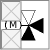
VISUALIZATION Icon_ML_AB_Up  // 50x50
VAR_INPUT
    ITF_STELLANTRIEB_IN   :   ITF_STELLANTRIEB;	
END_VAR
    Frame (4,16 18x18)
        shows Motor(ITF_STELLANTRIEB_IN := ITF_STELLANTRIEB_IN)
    Frame (20,9 24x32)
        shows ML_Ventil_AB_Up(rProzent := ITF_STELLANTRIEB_IN.proOnY)
    Image (1,1 20x20), invisible if: NOT ITF_STELLANTRIEB_IN.proIsWarning, image: CtaVisSymbols.ImagePool.CtaWarning
    Image (1,29 20x20), invisible if: NOT ITF_STELLANTRIEB_IN.proIsHandOnOrOff, image: CtaVisSymbols.ImagePool.front_hand_Yellow
    Image (1,29 20x20), invisible if: NOT ITF_STELLANTRIEB_IN.proHandOff, image: CtaVisSymbols.ImagePool.front_hand_Yellow_Off
END_VISUALIZATION

// 40 Visualizations/ICON/StellAntrieb_BASE/Icons/Motor_Left/Icon_ML_Verteiler
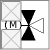
VISUALIZATION Icon_ML_Verteiler  // 50x50
VAR_INPUT
    ITF_STELLANTRIEB_IN   :   ITF_STELLANTRIEB;	
END_VAR
    Frame (4,16 18x18)
        shows Motor(ITF_STELLANTRIEB_IN := ITF_STELLANTRIEB_IN)
    Frame (20,9 24x32)
        shows ML_Ventil_Verteiler(rProzent := ITF_STELLANTRIEB_IN.proOnY)
    Image (1,1 20x20), invisible if: NOT ITF_STELLANTRIEB_IN.proIsWarning, image: CtaVisSymbols.ImagePool.CtaWarning
    Image (1,29 20x20), invisible if: NOT ITF_STELLANTRIEB_IN.proIsHandOnOrOff, image: CtaVisSymbols.ImagePool.front_hand_Yellow
    Image (1,29 20x20), invisible if: NOT ITF_STELLANTRIEB_IN.proHandOff, image: CtaVisSymbols.ImagePool.front_hand_Yellow_Off
END_VISUALIZATION

// 40 Visualizations/ICON/StellAntrieb_BASE/Icons/Motor_Left/Icon_ML_Durchfluss
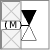
VISUALIZATION Icon_ML_Durchfluss  // 50x50
VAR_INPUT
    ITF_STELLANTRIEB_IN   :   ITF_STELLANTRIEB;	
END_VAR
    Frame (4,16 18x18)
        shows Motor(ITF_STELLANTRIEB_IN := ITF_STELLANTRIEB_IN)
    Frame (20,9 17x32)
        shows ML_Durchgang(rProzent := ITF_STELLANTRIEB_IN.proOnY)
    Image (1,1 20x20), invisible if: NOT ITF_STELLANTRIEB_IN.proIsWarning, image: CtaVisSymbols.ImagePool.CtaWarning
    Image (1,29 20x20), invisible if: NOT ITF_STELLANTRIEB_IN.proIsHandOnOrOff, image: CtaVisSymbols.ImagePool.front_hand_Yellow
    Image (1,29 20x20), invisible if: NOT ITF_STELLANTRIEB_IN.proHandOff, image: CtaVisSymbols.ImagePool.front_hand_Yellow_Off
END_VISUALIZATION

// 40 Visualizations/ICON/StellAntrieb_BASE/Icons/Motor_Right/Icon_MR_AB_Down
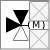
VISUALIZATION Icon_MR_AB_Down  // 50x50
VAR_INPUT
    ITF_STELLANTRIEB_IN   :   ITF_STELLANTRIEB;	
END_VAR
    Frame (27,16 18x18)
        shows Motor(ITF_STELLANTRIEB_IN := ITF_STELLANTRIEB_IN)
    Frame (5,9 24x32)
        shows MR_Ventil_AB_Down(rProzent := ITF_STELLANTRIEB_IN.proOnY)
    Image (29,1 20x20), invisible if: NOT ITF_STELLANTRIEB_IN.proIsWarning, image: CtaVisSymbols.ImagePool.CtaWarning
    Image (29,29 20x20), invisible if: NOT ITF_STELLANTRIEB_IN.proIsHandOnOrOff, image: CtaVisSymbols.ImagePool.front_hand_Yellow
    Image (29,29 20x20), invisible if: NOT ITF_STELLANTRIEB_IN.proHandOff, image: CtaVisSymbols.ImagePool.front_hand_Yellow_Off
END_VISUALIZATION

// 40 Visualizations/ICON/StellAntrieb_BASE/Icons/Motor_Right/Icon_MR_AB_Up
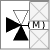
VISUALIZATION Icon_MR_AB_Up  // 50x50
VAR_INPUT
    ITF_STELLANTRIEB_IN   :   ITF_STELLANTRIEB;	
END_VAR
    Frame (27,16 18x18)
        shows Motor(ITF_STELLANTRIEB_IN := ITF_STELLANTRIEB_IN)
    Frame (5,9 24x32)
        shows MR_Ventil_AB_Up(rProzent := ITF_STELLANTRIEB_IN.proOnY)
    Image (29,1 20x20), invisible if: NOT ITF_STELLANTRIEB_IN.proIsWarning, image: CtaVisSymbols.ImagePool.CtaWarning
    Image (29,29 20x20), invisible if: NOT ITF_STELLANTRIEB_IN.proIsHandOnOrOff, image: CtaVisSymbols.ImagePool.front_hand_Yellow
    Image (29,29 20x20), invisible if: NOT ITF_STELLANTRIEB_IN.proHandOff, image: CtaVisSymbols.ImagePool.front_hand_Yellow_Off
END_VISUALIZATION

// 40 Visualizations/ICON/StellAntrieb_BASE/Icons/Motor_Right/Icon_MR_Durchfluss
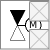
VISUALIZATION Icon_MR_Durchfluss  // 50x50
VAR_INPUT
    ITF_STELLANTRIEB_IN   :   ITF_STELLANTRIEB;	
END_VAR
    Frame (24,16 18x18)
        shows Motor(ITF_STELLANTRIEB_IN := ITF_STELLANTRIEB_IN)
    Frame (9,9 17x32)
        shows MR_Durchgang(rProzent := ITF_STELLANTRIEB_IN.proOnY)
    Image (29,1 20x20), invisible if: NOT ITF_STELLANTRIEB_IN.proIsWarning, image: CtaVisSymbols.ImagePool.CtaWarning
    Image (29,29 20x20), invisible if: NOT ITF_STELLANTRIEB_IN.proIsHandOnOrOff, image: CtaVisSymbols.ImagePool.front_hand_Yellow
    Image (29,29 20x20), invisible if: NOT ITF_STELLANTRIEB_IN.proHandOff, image: CtaVisSymbols.ImagePool.front_hand_Yellow_Off
END_VISUALIZATION

// 40 Visualizations/ICON/StellAntrieb_BASE/Icons/Motor_Right/Icon_MR_Verteiler
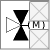
VISUALIZATION Icon_MR_Verteiler  // 50x50
VAR_INPUT
    ITF_STELLANTRIEB_IN   :   ITF_STELLANTRIEB;	
END_VAR
    Frame (27,16 18x18)
        shows Motor(ITF_STELLANTRIEB_IN := ITF_STELLANTRIEB_IN)
    Frame (5,9 24x32)
        shows MR_Ventil_Verteiler(rProzent := ITF_STELLANTRIEB_IN.proOnY)
    Image (29,1 20x20), invisible if: NOT ITF_STELLANTRIEB_IN.proIsWarning, image: CtaVisSymbols.ImagePool.CtaWarning
    Image (29,29 20x20), invisible if: NOT ITF_STELLANTRIEB_IN.proIsHandOnOrOff, image: CtaVisSymbols.ImagePool.front_hand_Yellow
    Image (29,29 20x20), invisible if: NOT ITF_STELLANTRIEB_IN.proHandOff, image: CtaVisSymbols.ImagePool.front_hand_Yellow_Off
END_VISUALIZATION

// 40 Visualizations/ICON/StellAntrieb_BASE/Icons/Motor_Above/Icon_MA_AB_L
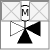
VISUALIZATION Icon_MA_AB_L  // 50x50
VAR_INPUT
    ITF_STELLANTRIEB_IN   :   ITF_STELLANTRIEB;	
END_VAR
    Frame (16,4 18x18)
        shows Motor(ITF_STELLANTRIEB_IN := ITF_STELLANTRIEB_IN)
    Frame (9,20 32x24)
        shows MA_Ventil_AB_L(rProzent := ITF_STELLANTRIEB_IN.proOnY)
    Image (1,1 20x20), invisible if: NOT ITF_STELLANTRIEB_IN.proIsWarning, image: CtaVisSymbols.ImagePool.CtaWarning
    Image (29,1 20x20), invisible if: NOT ITF_STELLANTRIEB_IN.proIsHandOnOrOff, image: CtaVisSymbols.ImagePool.front_hand_Yellow
    Image (29,1 20x20), invisible if: NOT ITF_STELLANTRIEB_IN.proHandOff, image: CtaVisSymbols.ImagePool.front_hand_Yellow_Off
END_VISUALIZATION

// 40 Visualizations/ICON/StellAntrieb_BASE/Icons/Motor_Above/Icon_MA_AB_R
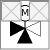
VISUALIZATION Icon_MA_AB_R  // 50x50
VAR_INPUT
    ITF_STELLANTRIEB_IN   :   ITF_STELLANTRIEB;	
END_VAR
    Frame (16,4 18x18)
        shows Motor(ITF_STELLANTRIEB_IN := ITF_STELLANTRIEB_IN)
    Frame (9,20 32x24)
        shows MA_Ventil_AB_R(rProzent := ITF_STELLANTRIEB_IN.proOnY)
    Image (1,1 20x20), invisible if: NOT ITF_STELLANTRIEB_IN.proIsWarning, image: CtaVisSymbols.ImagePool.CtaWarning
    Image (29,1 20x20), invisible if: NOT ITF_STELLANTRIEB_IN.proIsHandOnOrOff, image: CtaVisSymbols.ImagePool.front_hand_Yellow
    Image (29,1 20x20), invisible if: NOT ITF_STELLANTRIEB_IN.proHandOff, image: CtaVisSymbols.ImagePool.front_hand_Yellow_Off
END_VISUALIZATION

// 40 Visualizations/ICON/StellAntrieb_BASE/Icons/Motor_Above/Icon_MA_Durchfluss
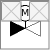
VISUALIZATION Icon_MA_Durchfluss  // 50x50
VAR_INPUT
    ITF_STELLANTRIEB_IN   :   ITF_STELLANTRIEB;	
END_VAR
    Frame (16,4 18x18)
        shows Motor(ITF_STELLANTRIEB_IN := ITF_STELLANTRIEB_IN)
    Frame (9,20 32x17)
        shows MA_Durchgang(rProzent := ITF_STELLANTRIEB_IN.proOnY)
    Image (1,1 20x20), invisible if: NOT ITF_STELLANTRIEB_IN.proIsWarning, image: CtaVisSymbols.ImagePool.CtaWarning
    Image (29,1 20x20), invisible if: NOT ITF_STELLANTRIEB_IN.proIsHandOnOrOff, image: CtaVisSymbols.ImagePool.front_hand_Yellow
    Image (29,1 20x20), invisible if: NOT ITF_STELLANTRIEB_IN.proHandOff, image: CtaVisSymbols.ImagePool.front_hand_Yellow_Off
END_VISUALIZATION

// 40 Visualizations/ICON/StellAntrieb_BASE/Icons/Motor_Above/Icon_MA_Verteiler
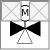
VISUALIZATION Icon_MA_Verteiler  // 50x50
VAR_INPUT
    ITF_STELLANTRIEB_IN   :   ITF_STELLANTRIEB;	
END_VAR
    Frame (16,4 18x18)
        shows Motor(ITF_STELLANTRIEB_IN := ITF_STELLANTRIEB_IN)
    Frame (9,20 32x24)
        shows MA_Ventil_Verteiler(rProzent := ITF_STELLANTRIEB_IN.proOnY)
    Image (1,1 20x20), invisible if: NOT ITF_STELLANTRIEB_IN.proIsWarning, image: CtaVisSymbols.ImagePool.CtaWarning
    Image (29,1 20x20), invisible if: NOT ITF_STELLANTRIEB_IN.proIsHandOnOrOff, image: CtaVisSymbols.ImagePool.front_hand_Yellow
    Image (29,1 20x20), invisible if: NOT ITF_STELLANTRIEB_IN.proHandOff, image: CtaVisSymbols.ImagePool.front_hand_Yellow_Off
END_VISUALIZATION

// 40 Visualizations/ICON/StellAntrieb_BASE/Icons/Motor_Below/Icon_MB_AB_L
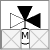
VISUALIZATION Icon_MB_AB_L  // 50x50
VAR_INPUT
    ITF_STELLANTRIEB_IN   :   ITF_STELLANTRIEB;	
END_VAR
    Frame (16,27 18x18)
        shows Motor(ITF_STELLANTRIEB_IN := ITF_STELLANTRIEB_IN)
    Frame (9,5 32x24)
        shows MB_Ventil_AB_L(rProzent := ITF_STELLANTRIEB_IN.proOnY)
    Image (1,29 20x20), invisible if: NOT ITF_STELLANTRIEB_IN.proIsWarning, image: CtaVisSymbols.ImagePool.CtaWarning
    Image (29,29 20x20), invisible if: NOT ITF_STELLANTRIEB_IN.proIsHandOnOrOff, image: CtaVisSymbols.ImagePool.front_hand_Yellow
    Image (29,29 20x20), invisible if: NOT ITF_STELLANTRIEB_IN.proHandOff, image: CtaVisSymbols.ImagePool.front_hand_Yellow_Off
END_VISUALIZATION

// 40 Visualizations/ICON/StellAntrieb_BASE/Icons/Motor_Below/Icon_MB_AB_R
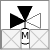
VISUALIZATION Icon_MB_AB_R  // 50x50
VAR_INPUT
    ITF_STELLANTRIEB_IN   :   ITF_STELLANTRIEB;	
END_VAR
    Frame (16,27 18x18)
        shows Motor(ITF_STELLANTRIEB_IN := ITF_STELLANTRIEB_IN)
    Frame (9,5 32x24)
        shows MB_Ventil_AB_R(rProzent := ITF_STELLANTRIEB_IN.proOnY)
    Image (1,29 20x20), invisible if: NOT ITF_STELLANTRIEB_IN.proIsWarning, image: CtaVisSymbols.ImagePool.CtaWarning
    Image (29,29 20x20), invisible if: NOT ITF_STELLANTRIEB_IN.proIsHandOnOrOff, image: CtaVisSymbols.ImagePool.front_hand_Yellow
    Image (29,29 20x20), invisible if: NOT ITF_STELLANTRIEB_IN.proHandOff, image: CtaVisSymbols.ImagePool.front_hand_Yellow_Off
END_VISUALIZATION

// 40 Visualizations/ICON/StellAntrieb_BASE/Icons/Motor_Below/Icon_MB_Verteiler
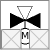
VISUALIZATION Icon_MB_Verteiler  // 50x50
VAR_INPUT
    ITF_STELLANTRIEB_IN   :   ITF_STELLANTRIEB;	
END_VAR
    Frame (16,27 18x18)
        shows Motor(ITF_STELLANTRIEB_IN := ITF_STELLANTRIEB_IN)
    Frame (9,5 32x24)
        shows MB_Ventil_Verteiler(rProzent := ITF_STELLANTRIEB_IN.proOnY)
    Image (1,29 20x20), invisible if: NOT ITF_STELLANTRIEB_IN.proIsWarning, image: CtaVisSymbols.ImagePool.CtaWarning
    Image (29,29 20x20), invisible if: NOT ITF_STELLANTRIEB_IN.proIsHandOnOrOff, image: CtaVisSymbols.ImagePool.front_hand_Yellow
    Image (29,29 20x20), invisible if: NOT ITF_STELLANTRIEB_IN.proHandOff, image: CtaVisSymbols.ImagePool.front_hand_Yellow_Off
END_VISUALIZATION

// 40 Visualizations/ICON/StellAntrieb_BASE/Icons/Motor_Below/Icon_MB_Durchfluss
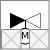
VISUALIZATION Icon_MB_Durchfluss  // 50x50
VAR_INPUT
    ITF_STELLANTRIEB_IN   :   ITF_STELLANTRIEB;	
END_VAR
    Frame (16,27 18x18)
        shows Motor(ITF_STELLANTRIEB_IN := ITF_STELLANTRIEB_IN)
    Frame (9,12 32x17)
        shows MB_Durchgang(rProzent := ITF_STELLANTRIEB_IN.proOnY)
    Image (1,29 20x20), invisible if: NOT ITF_STELLANTRIEB_IN.proIsWarning, image: CtaVisSymbols.ImagePool.CtaWarning
    Image (29,29 20x20), invisible if: NOT ITF_STELLANTRIEB_IN.proIsHandOnOrOff, image: CtaVisSymbols.ImagePool.front_hand_Yellow
    Image (29,29 20x20), invisible if: NOT ITF_STELLANTRIEB_IN.proHandOff, image: CtaVisSymbols.ImagePool.front_hand_Yellow_Off
END_VISUALIZATION

// 40 Visualizations/ICON/StellAntrieb_RIGHT/Motor_Right/Valve_AB_Down/Below/StellAntrieb_MR_Valve_AB_Down_Txt_R_Below
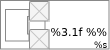
VISUALIZATION StellAntrieb_MR_Valve_AB_Down_Txt_R_Below  // 110x50
VAR_INPUT
    ITF_STELLANTRIEB_IN   	:   ITF_STELLANTRIEB;	
END_VAR
VAR_INPUT CONSTANT
	stExklParameter			:	STRING[40] := '';
END_VAR
VAR CONSTANT
	uiIconNr				: 	UINT := 25;
END_VAR
    Frame (0,0 110x50), invisible if: NOT fcCheckQuerryReturnIcon(_ITF_In := ITF_STELLANTRIEB_IN,_uiIconNr_In := uiIconNr)
        shows StellAntrieb_MR_Valve_AB_Down_RB_CheckQuerry(ITF_STELLANTRIEB_IN := ITF_STELLANTRIEB_IN, stExklParameter := stExklParameter)
        shows Icon()
END_VISUALIZATION

// 40 Visualizations/ICON/StellAntrieb_RIGHT/Motor_Right/Valve_AB_Down/Below/StellAntrieb_MR_Valve_AB_Down_RB_CheckEnabled
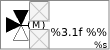
VISUALIZATION StellAntrieb_MR_Valve_AB_Down_RB_CheckEnabled  // 110x50
VAR_INPUT
    ITF_STELLANTRIEB_IN   	:   ITF_STELLANTRIEB;
	stExklParameter			:	STRING[40];
END_VAR
    Frame (0,0 50x50), invisible if: NOT ITF_STELLANTRIEB_IN.proIsEnabled
        shows Icon_MR_AB_Down(ITF_STELLANTRIEB_IN := ITF_STELLANTRIEB_IN)
    Frame (50,25 60x25), invisible if: NOT ITF_STELLANTRIEB_IN.proIsEnabled
        shows ValueDwnUp(ITF_STELLANTRIEB_IN := ITF_STELLANTRIEB_IN, uiTextAusrichtung := 4)
    Rectangle (0,0 110x50)
        OnMouseClick:  Dialog=StellAntrieb_POPUP, Parameters={stExklParameter: stExklParameter, ITF_STELLANTRIEBIN: ITF_STELLANTRIEB_IN, uiPopUpGruppe: 0}, OpenCentered=True
END_VISUALIZATION

// 40 Visualizations/ICON/StellAntrieb_RIGHT/Motor_Right/Valve_AB_Down/Below/StellAntrieb_MR_Valve_AB_Down_RB_CheckQuerry
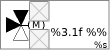
VISUALIZATION StellAntrieb_MR_Valve_AB_Down_RB_CheckQuerry  // 110x50
VAR_INPUT
    ITF_STELLANTRIEB_IN   	:   ITF_STELLANTRIEB;	
	stExklParameter			:	STRING[40];
END_VAR
    Frame (0,0 110x50)
        shows StellAntrieb_MR_Valve_AB_Down_RB_CheckEnabled(ITF_STELLANTRIEB_IN := ITF_STELLANTRIEB_IN, stExklParameter := stExklParameter)
END_VISUALIZATION

// 40 Visualizations/ICON/StellAntrieb_LEFT/Motor_LEFT/Valve_AB_Down/Above/StellAntrieb_ML_Valve_AB_Down_LA_CheckEnabled
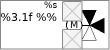
VISUALIZATION StellAntrieb_ML_Valve_AB_Down_LA_CheckEnabled  // 110x50
VAR_INPUT
    ITF_STELLANTRIEB_IN   	:   ITF_STELLANTRIEB;	
	stExklParameter			:	STRING[40];
END_VAR
    Frame (61,0 50x50), invisible if: NOT ITF_STELLANTRIEB_IN.proIsEnabled
        shows Icon_ML_AB_Down(ITF_STELLANTRIEB_IN := ITF_STELLANTRIEB_IN)
    Frame (0,0 60x25), invisible if: NOT ITF_STELLANTRIEB_IN.proIsEnabled
        shows ValueUpDwn(ITF_STELLANTRIEB_IN := ITF_STELLANTRIEB_IN, uiTextAusrichtung := 6)
    Rectangle (0,0 110x50)
        OnMouseClick:  Dialog=StellAntrieb_POPUP, Parameters={stExklParameter: stExklParameter, ITF_STELLANTRIEBIN: ITF_STELLANTRIEB_IN, uiPopUpGruppe: 0}, OpenCentered=True
END_VISUALIZATION

// 40 Visualizations/ICON/StellAntrieb_LEFT/Motor_LEFT/Valve_AB_Down/Above/StellAntrieb_ML_Valve_AB_Down_LA_CheckQuerry
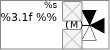
VISUALIZATION StellAntrieb_ML_Valve_AB_Down_LA_CheckQuerry  // 110x50
VAR_INPUT
    ITF_STELLANTRIEB_IN   	:   ITF_STELLANTRIEB;
	stExklParameter			:	STRING[40];
END_VAR
    Frame (0,0 110x50)
        shows StellAntrieb_ML_Valve_AB_Down_LA_CheckEnabled(ITF_STELLANTRIEB_IN := ITF_STELLANTRIEB_IN, stExklParameter := stExklParameter)
END_VISUALIZATION

// 40 Visualizations/ICON/StellAntrieb_LEFT/Motor_LEFT/Valve_AB_Down/Above/StellAntrieb_ML_Valve_AB_Down_Txt_L_Above
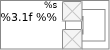
VISUALIZATION StellAntrieb_ML_Valve_AB_Down_Txt_L_Above  // 110x50
VAR_INPUT
    ITF_STELLANTRIEB_IN   	:   ITF_STELLANTRIEB;	
END_VAR
VAR_INPUT CONSTANT
	stExklParameter			:	STRING[40] := '';
END_VAR
VAR CONSTANT
	uiIconNr				: 	UINT := 8;
END_VAR
    Frame (0,0 110x50), invisible if: NOT fcCheckQuerryReturnIcon(_ITF_In := ITF_STELLANTRIEB_IN,_uiIconNr_In := uiIconNr)
        shows StellAntrieb_ML_Valve_AB_Down_LA_CheckQuerry(ITF_STELLANTRIEB_IN := ITF_STELLANTRIEB_IN, stExklParameter := stExklParameter)
        shows Icon()
END_VISUALIZATION

// 40 Visualizations/ICON/StellAntrieb_LEFT/Motor_LEFT/Valve_AB_Down/Below/StellAntrieb_ML_Valve_AB_Down_LB_CheckEnabled
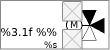
VISUALIZATION StellAntrieb_ML_Valve_AB_Down_LB_CheckEnabled  // 110x50
VAR_INPUT
    ITF_STELLANTRIEB_IN   	:   ITF_STELLANTRIEB;
	stExklParameter			:	STRING[40];
END_VAR
    Frame (61,0 50x50), invisible if: NOT ITF_STELLANTRIEB_IN.proIsEnabled
        shows Icon_ML_AB_Down(ITF_STELLANTRIEB_IN := ITF_STELLANTRIEB_IN)
    Frame (0,25 60x25), invisible if: NOT ITF_STELLANTRIEB_IN.proIsEnabled
        shows ValueDwnUp(ITF_STELLANTRIEB_IN := ITF_STELLANTRIEB_IN, uiTextAusrichtung := 6)
    Rectangle (0,0 110x50)
        OnMouseClick:  Dialog=StellAntrieb_POPUP, Parameters={stExklParameter: stExklParameter, ITF_STELLANTRIEBIN: ITF_STELLANTRIEB_IN, uiPopUpGruppe: 0}, OpenCentered=True
END_VISUALIZATION

// 40 Visualizations/ICON/StellAntrieb_LEFT/Motor_LEFT/Valve_AB_Down/Below/StellAntrieb_ML_Valve_AB_Down_LB_CheckQuerry
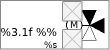
VISUALIZATION StellAntrieb_ML_Valve_AB_Down_LB_CheckQuerry  // 110x50
VAR_INPUT
    ITF_STELLANTRIEB_IN   	:   ITF_STELLANTRIEB;
	stExklParameter			:	STRING[40];
END_VAR
    Frame (0,0 110x50)
        shows StellAntrieb_ML_Valve_AB_Down_LB_CheckEnabled(ITF_STELLANTRIEB_IN := ITF_STELLANTRIEB_IN, stExklParameter := stExklParameter)
END_VISUALIZATION

// 40 Visualizations/ICON/StellAntrieb_LEFT/Motor_LEFT/Valve_AB_Down/Below/StellAntrieb_ML_Valve_AB_Down_Txt_L_Below
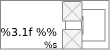
VISUALIZATION StellAntrieb_ML_Valve_AB_Down_Txt_L_Below  // 110x50
VAR_INPUT
    ITF_STELLANTRIEB_IN   	:   ITF_STELLANTRIEB;	
END_VAR
VAR_INPUT CONSTANT
	stExklParameter			:	STRING[40] := '';
END_VAR
VAR CONSTANT
	uiIconNr				: 	UINT := 9;
END_VAR
    Frame (0,0 110x50), invisible if: NOT fcCheckQuerryReturnIcon(_ITF_In := ITF_STELLANTRIEB_IN,_uiIconNr_In := uiIconNr)
        shows StellAntrieb_ML_Valve_AB_Down_LB_CheckQuerry(ITF_STELLANTRIEB_IN := ITF_STELLANTRIEB_IN, stExklParameter := stExklParameter)
        shows Icon()
END_VISUALIZATION

// 40 Visualizations/ICON/StellAntrieb_RIGHT/Motor_Below/Valve_AB_Left/StellAntrieb_MB_Valve_AB_Left_RB_CheckEnabled
